ABB RobotStudio station: parte0.rsstn

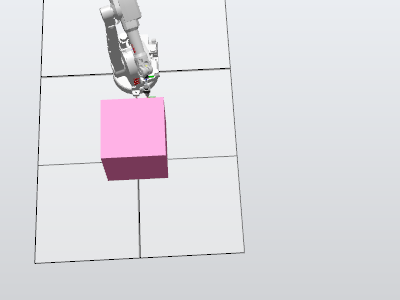
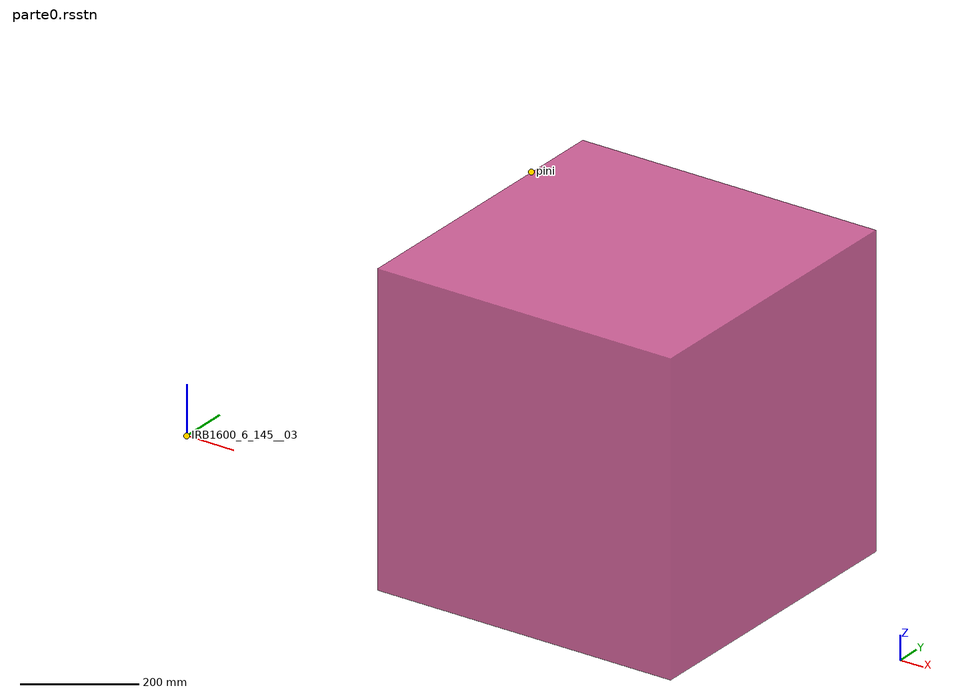
[picture v1: parts stored in the station drawn from their meshes, with robot base, taught points and paths (robot models come from the ABB library and are not in the file)]
Station parte0 (saved by RobotStudio 24.1.10713.1)
Controller Controlador3
  mechanical unit ROB_1: IRB1600_6_145__03, 6 joints, base frame (0, 0, 0) mm
Layout (positions relative to the parent item):
  - IRB1600_6_145__03 [mechanism, from %ABB.RobotStudio.Models.IRB1600%\IRB1600_6_145_G_03.rslib] at (0, 0, 0) mm; joint values [0.326, -0.2862, 0.8219, -0.4788, 0.4423, 0.699] (rad or m)
  - MyTool [mechanism, from Training Objects\myTool.rslib] at (483.67, 150, 800.53) mm, rotated rx -180 ry 38 rz -180 deg
  - Pieza_1 [part], size 600 x 600 x 600 mm
Attachment: MyTool is attached to IRB1600_6_145__03 / Link6
Targets, tools, work objects and paths stored in the station, written as RAPID:
! task T_ROB1
MODULE CalibData
  PERS tooldata MyTool:=[TRUE,[[31.792631019,0,229.638935148],[0.945518576,0,0.325568154,0]],[1,[0,0,1],[1,0,0,0],0,0,0]];
ENDMODULE

! task T_ROB1
MODULE Module1
  CONST robtarget pini:=[[600,150,600],[0,0,1,0],[0,0,0,0],[9E+09,9E+09,9E+09,9E+09,9E+09,9E+09]];
  PROC Path_10()
    MoveL pini,v1000,z100,MyTool\WObj:=wobj0;
  ENDPROC
  PROC main()
  ENDPROC
ENDMODULE

